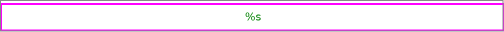
VISUALIZATION MessageBox_1  // 504x32
VAR_IN_OUT
	message_1 : ST_MessageBoxText;
END_VAR
    Textfield (3,2 500x30), "%s", text variable: message_1.sText
        p55702900: message_1.nColor
    Rectangle (0,3 504x28)
        p3450524324: message_1.nColor
END_VISUALIZATION

(* stored: Version 1.1.0.1
   Visu MessageBox_1: Id {fd934f34-0f64-4f0f-8369-f9ad9a65d52c} *)
